PROGRAM GetPreviousLine

VAR_OUTPUT
	arrRecords: ST_ProgramStruct;
	sSeverity: WSTRING(255);
	bError :BOOL;

	iLines: UDINT;
END_VAR
VAR
	STProgram: ST_ProgramStruct;
	now : TIMESTRUCT;
	nowMinutes : LINT;
	
	previousMinute: LINT;

	

	
	fbPLCDBRead : FB_PLCDBRead(sNetID:='',tTimeout:=T#5S);
	fbSqlCommand : FB_SQLCommand(sNetID := '', tTimeout := T#5S);
	
	
	intTime: DINT;
	todTime: TOD;

	sCmd: STRING(255);

	dIntSqlResult: DINT;
	fbSQLDatabase: FB_SQLDatabase(sNetID:='', tTimeout:=T#10S);
	fbSQLResult: FB_SQLResult(sNetID:='', tTimeout:=T#10S);
	result: I_TcResultEvent;


	iState: INT;
	fbTON: TON := (PT := TIME#10s0ms);

END_VAR

//Build command


now := GVL.fbLocalSystemTime.systemTime;
nowMinutes := now.wHour*60+now.wMinute;



sCmd :=CONCAT('SELECT  *  FROM [Programs]  WHERE [ProgramNameID]=',LINT_TO_STRING(GVL.CurrentProgram));

sCmd :=CONCAT(sCmd,' AND [time] <=');

sCmd := CONCAT(sCMD,LINT_TO_STRING(nowMinutes));

sCmd:= CONCAT(sCMD,' ORDER BY [time] DESC');
//State machine
CASE iState OF
0:
//IDLE
fbTON();
IF fbTON.Q=TRUE THEN
	iState:=1;
	fbTON.IN:=FALSE;
	bError := FALSE; 
ELSE
	fbTON.IN:=TRUE;
END_IF
//Connect
1:
	IF fbSqlDatabase.Connect(1) THEN
		IF fbSqlDatabase.bError THEN
			iState := 255;
			result := fbSqlDatabase.ipTcResultEvent;
			sSeverity := result.Text;
			bError := TRUE; 		
		ELSE
			//If sucessful, point the connection to the sql command function
			fbSqlDatabase.CreateCmd(ADR(fbSqlCommand));
			iState := 2;
		END_IF
	END_IF
2:
//Send the sql command
	IF fbSQLCommand.ExecuteDataReturn(ADR(sCmd), SIZEOF(sCmd), ADR(fbSqlResult)) THEN
		IF fbSQLCommand.bError THEN
			iState := 255;
			result := fbSQLCommand.ipTcResultEvent;
			sSeverity := result.Text;
			bError := TRUE;
		ELSE
			iState := 3; 
			iLines:=fbSqlResult.nDataCount;
		END_IF
	END_IF
		
3:
//Read the sql result
	IF fbSqlResult.Read(0, 1, ADR(arrRecords), SIZEOF(arrRecords), TRUE, TRUE) THEN
		IF fbSqlResult.bError THEN
			result := fbSqlResult.ipTcResultEvent;
			sSeverity := result.Text;
			iState:=255;
			bError := TRUE;
		ELSE 
			iState:=4;
			
			result := fbSqlResult.ipTcResultEvent;
			sSeverity := result.Text;
		END_IF
	

	END_IF
4:
	IF 	fbSqlDatabase.Disconnect() THEN
		bError := FALSE;
		iState:=0;
	END_IF
255:
	IF 	fbSqlDatabase.Disconnect() THEN
		iState:=0;	
		bError := TRUE;
		result := fbSqlResult.ipTcResultEvent;
		sSeverity := result.Text;
	END_IF
	
END_CASE

END_PROGRAM

(* stored: Version 1.1.0.1, ProductVersion 3.1.4022.16
   POU GetPreviousLine: Id {fb22217d-049e-421e-9117-44d2b1dc44b0}, SpecialFunc None *)
